% RSLogix 500 project carP.RSS, saved by version 8.30.00.15 %
PROJECT "UNTITLED"    % processor: MicroLogix 1400 %

PROGRAM FILES
  LAD 2   7 rungs

DATA FILES
  O0 OUTPUT  6 elements
  I1 INPUT  8 elements
  S2 STATUS  66 elements
  B3 BINARY  1 elements
  T4 TIMER  1 elements
  C5 COUNTER  1 elements
  R6 CONTROL  1 elements
  N7 INTEGER  7 elements
  F8 FLOAT  1 elements

LADDER 2
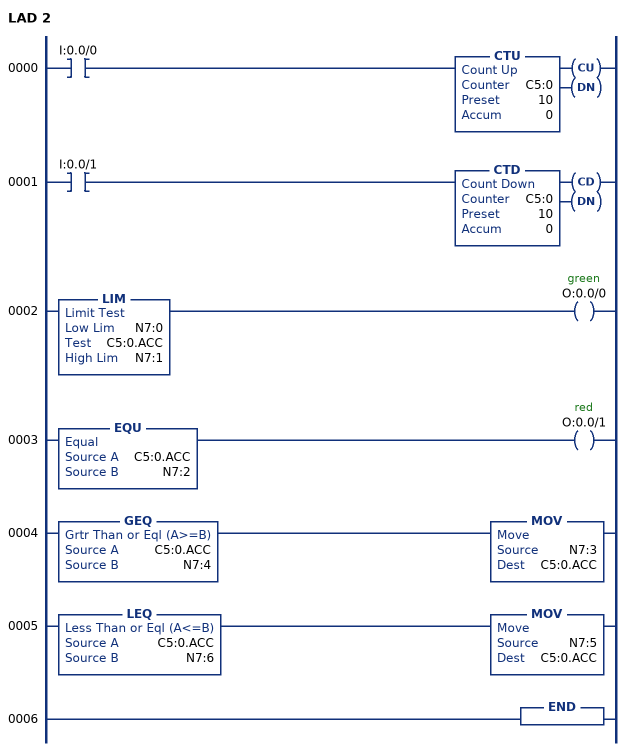
% Rung: 0 %
SOR XIC I:0.0/0 CTU C5:0 10 0 EOR
% Rung: 1 %
SOR XIC I:0.0/1 CTD C5:0 10 0 EOR
% Rung: 2 %
SOR LIM N7:0 C5:0.ACC N7:1 OTE O:0.0/0 EOR
%   O:0.0/0  "green" %
% Rung: 3 %
SOR EQU C5:0.ACC N7:2 OTE O:0.0/1 EOR
%   O:0.0/1  "red" %
% Rung: 4 %
SOR GEQ C5:0.ACC N7:4 MOV N7:3 C5:0.ACC EOR
% Rung: 5 %
SOR LEQ C5:0.ACC N7:6 MOV N7:5 C5:0.ACC EOR
%   N7:6  N7 %
% Rung: 6 %
SOR END EOR

DATA TABLE (non-zero values as saved)
DATA C5
% .PRE .ACC %
% C5:0 % 10 0
DATA N7
% N7:0 % 0 9 10 10 10 0 0
